INTERFACE I_Magnetventil

METHOD M_A_OEFFNEN : BOOL
VAR_INPUT
END_VAR
END_METHOD

METHOD M_A_SCHLIESSEN : BOOL
VAR_INPUT
END_VAR
END_METHOD

METHOD M_M_OEFFNEN : BOOL
VAR_INPUT
END_VAR
END_METHOD

METHOD M_M_SCHLIESSEN : BOOL
VAR_INPUT
END_VAR
END_METHOD

PROPERTY P_Status : INT
GET
END_GET
END_PROPERTY

END_INTERFACE

(* stored: Version 1.1.0.1, ProductVersion 3.1.4024.12
   Itf I_Magnetventil: Id {a17bf922-bf26-4dd4-85a2-f2356bfb708a}
   Method M_A_OEFFNEN: Id {fa812cba-d9ae-4232-b0bd-0aacf356e7a0}
   Method M_A_SCHLIESSEN: Id {96fa8735-fb03-460b-90ed-190789c8fb7c}
   Method M_M_OEFFNEN: Id {bc3072cc-c19f-4ad0-a0a3-0b54b2223672}
   Method M_M_SCHLIESSEN: Id {ccf9c1a0-1761-4444-8cdc-e453baac0299}
   Property P_Status: Id {801f1074-6e96-4281-b554-66700cd46471}
   Get Get: Id {e5353621-4ed4-4fc9-8ca8-1d0392b65a59} *)
